// TIA Portal V19 export
TYPE "IFM_TA1612_IO"
   STRUCT
      Addr : Int;   // IO Address
      Value : Real;   // Temperature_C
      OL : Bool;   // value over range
      UL : Bool;   // value under reange
      O_DI4 : Bool;   // Port pin 4
      O_DI2 : Bool;   // Port pin 2
      O_DA : Bool;   // Device Attached
      O_DE : Bool;   // Device Error
      O_PQ : Bool;   // Value Valid
   END_STRUCT;
END_TYPE
